ABB RobotStudio station: p3_Ejercicio_2018.rspag

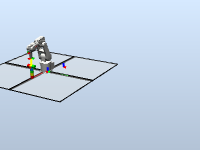
--- station ---
Station p3_Ejercicio_2018 (saved by RobotStudio 6.6.7701.1025)
Controller Sistema8
  mechanical unit ROB_1: IRB120_3_58__01_2, 6 joints, base frame (0, 0, 0) mm
Layout (positions relative to the parent item):
  - Grupo_1 [graphiccomponentgroup]
    - Pieza4 [part] at (170.19, 192.84, 150.02) mm, rotated rx 0 ry 0 rz -40 deg
    - Pieza3_2 [part] at (99.94, 75, 235.51) mm, rotated rx 90 ry 2 rz 0 deg
    - Pieza3 [part] at (100, 0, 100) mm
    - Pieza2_2 [part] at (99.94, 25, 235.51) mm, rotated rx 90 ry 2 rz 0 deg
    - Pieza2 [part] at (100, 0, 50.05) mm
    - Pieza1_2 [part] at (99.94, -25, 235.51) mm, rotated rx 90 ry 2 rz 0 deg
    - Pieza1 [part] at (100, 0, 0.18) mm
  - IRB120_3_58__01_2 [mechanism, from Robots\IRB120_3_58_G_01.rslib] at (0, 0, 0) mm; joint values [0, 0.3398, -0.1178, 0, 1.3488, 3.1416] (rad or m)
  - SC_Ventosa2 [smart component]
      signals: DI vacio, DI soplado, DO Vacuostato
      connections:
        SC_Ventosa.Vacuostato -> SC_Ventosa2.Vacuostato
        SC_Ventosa2.vacio -> SC_Ventosa.vacio
        SC_Ventosa2.soplado -> SC_Ventosa.soplado
    - SC_Ventosa [smart component] at (0, 0, 0) mm
        signals: DI vacio, DI soplado, DO Vacuostato
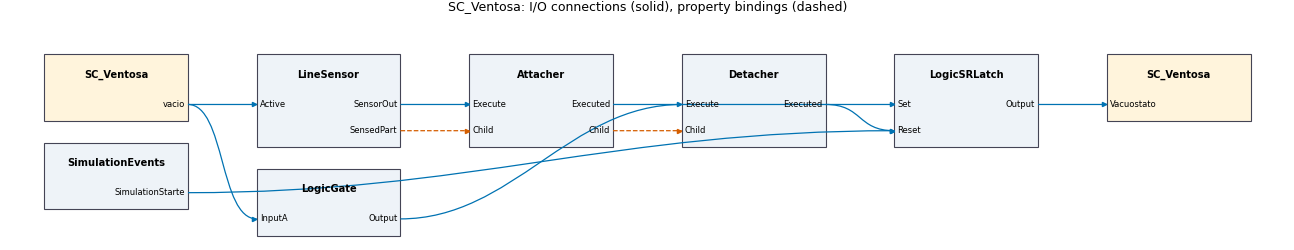
        connections:
          SC_Ventosa.vacio -> LineSensor.Active
          LineSensor.SensorOut -> Attacher.Execute
          Attacher.Executed -> LogicSRLatch.Set
          LogicSRLatch.Output -> SC_Ventosa.Vacuostato
          SC_Ventosa.vacio -> LogicGate.InputA
          LogicGate.Output -> Detacher.Execute
          Detacher.Executed -> LogicSRLatch.Reset
          SimulationEvents.SimulationStarted -> LogicSRLatch.Reset
          LineSensor.SensedPart => Attacher.Child
          Attacher.Child => Detacher.Child
      - MyNewTool [mechanism] at (400, 0, 474.33) mm, rotated rx -180 ry 0 rz 0 deg
          TCP Ventosa at (0, 0, 100) mm, rotated rx 180 ry 0 rz 0 deg
          links: Ventosa
      - LineSensor [smart component, from Components\LineSensor.rslib] at (400, 0, 474.33) mm, rotated rx -180 ry 0 rz 0 deg
          properties: Start=[0 0 0.0991]; End=[0 0 0.12]; Radius=0.002; SensedPart=Pieza1_2; SensedPoint=[0.4 -0.0750000686645508 0.231999969482422]
        - _sensorPart_ [part]
      - Attacher [smart component, from Components\Attacher.rslib]
          properties: Parent=MyNewTool; Flange=0; Child=Pieza1_2; Mount=false; Offset=[0 0 0]; Orientation=[0 0 0]
      - Detacher [smart component, from Components\Detacher.rslib]
          properties: Child=Pieza1_2; KeepPosition=true
      - LogicSRLatch [smart component, from Components\LogicSRLatch.rslib]
      - LogicGate [smart component, from Components\LogicGate.rslib]
          properties: Operator=NOT; Delay=0
      - SimulationEvents [smart component, from Components\SimulationEvents.rslib]
Attachment: MyNewTool is attached to IRB120_3_58__01_2 / Link6
Attachment: LineSensor is attached to MyNewTool / Ventosa
Station logic (signal -> signal, property => property):
  SC_Ventosa2.Vacuostato -> Sistema8.Vacuostado
  Sistema8.vacio -> SC_Ventosa2.vacio
  Sistema8.soplado -> SC_Ventosa2.soplado

--- Backups/Sistema8/RAPID/TASK1/PROGMOD/CalibData.mod ---
MODULE CalibData
	PERS tooldata Ventosa:=[TRUE,[[0.000043514,0,100],[0,1,0,-0.000000126]],[1,[0.000025299,0,100],[1,0,0,0],0,0,0]];
ENDMODULE

--- Backups/Sistema8/RAPID/TASK1/PROGMOD/Module1.mod ---
MODULE Module1
	CONST robtarget Target_10:=[[400.000012438,0,374.334869531],[1,0,-0.000000093,-0.000000044],[0,0,2,0],[9E+09,9E+09,9E+09,9E+09,9E+09,9E+09]];
	CONST robtarget Target_20:=[[400,0,200],[1,0,0,0],[0,0,1,0],[9E+09,9E+09,9E+09,9E+09,9E+09,9E+09]];
	CONST robtarget Target_30:=[[90.077,394.84,0],[1,0,0,0],[0,0,2,0],[9E+09,9E+09,9E+09,9E+09,9E+09,9E+09]];
    CONST robtarget Target_40:=[[-6.960015192,400.000008696,149.999960784],[0.694658412,0.000000021,-0.000000021,0.71933976],[1,-1,1,0],[9E+09,9E+09,9E+09,9E+09,9E+09,9E+09]];

	PROC Path_10()
        VAR robtarget reposo;
        VAR robtarget reposo1;
        VAR robtarget reposo2;
        VAR robtarget reposo3;
        VAR robtarget reposo4;

        VAR robtarget aux1;
        VAR robtarget aux2;
        VAR robtarget aux3;
        VAR robtarget aux4;




        reposo := Offs(Target_30,0,0,300);
        reposo1 := Offs(Target_30,0,0,50);
        reposo2 := Offs(Target_30,0,0,100);
        reposo3 := Offs(Target_30,0,0,150);
        reposo4 := Offs(Target_30,0,0,200);

        aux1 := Offs(Target_20,0,0,-50);
        aux2 := Offs(Target_20,0,0,-100);
        aux3 := Offs(Target_20,0,0,-150);
        aux4 := Offs(Target_20,0,0,-200);




        !Voy a inicio
	    MoveL Target_10,v1000,z100,Ventosa\WObj:=wobj0;
	    WaitTime 1;
        !Cojo la 1 pieza
	    MoveL Target_20,v1000,fine,Ventosa\WObj:=wobj0;
        WaitTime 1;
        SetDO vacio,1;
        WaitTime 1;
        !La dejo en posicion de reposo
        MoveJ reposo,v1000,fine,Ventosa\WObj:=wobj0;
	    MoveL reposo1,v500,fine,Ventosa\WObj:=wobj0;
        WaitTime 1;
	    SetDO vacio,0;
        WaitTime 1;
        !Vuelvo a inicio
        MoveJ Target_10,v1000,fine,Ventosa\WObj:=wobj0;

        !Cojo la 2 pieza
	    MoveL aux1,v1000,fine,Ventosa\WObj:=wobj0;
        WaitTime 1;
        SetDO vacio,1;
        WaitTime 1;
        !La dejo en posicion de reposo
        MoveJ reposo,v1000,fine,Ventosa\WObj:=wobj0;
	    MoveL reposo2,v500,fine,Ventosa\WObj:=wobj0;
	    SetDO vacio,0;
        WaitTime 1;
        !Vuelvo a inicio
        MoveJ Target_10,v1000,fine,Ventosa\WObj:=wobj0;

        !Cojo la 3 pieza
	    WaitTime 1;
	    MoveJ Target_10,v1000,fine,Ventosa\WObj:=wobj0;
	    MoveL aux2,v1000,fine,Ventosa\WObj:=wobj0;
        WaitTime 1;
        SetDO vacio,1;
        WaitTime 1;
        !La dejo en posicion de reposo
        MoveJ reposo,v1000,fine,Ventosa\WObj:=wobj0;
	    MoveL reposo3,v500,fine,Ventosa\WObj:=wobj0;
	    SetDO vacio,0;
        WaitTime 1;
        !Vuelvo a inicio
        MoveJ Target_10,v1000,fine,Ventosa\WObj:=wobj0;

        !Cojo la 4 pieza
	    MoveL aux3,v1000,fine,Ventosa\WObj:=wobj0;
        WaitTime 1;
        SetDO vacio,1;
        WaitTime 1;
        !La dejo en posicion de reposo
        MoveJ reposo,v1000,fine,Ventosa\WObj:=wobj0;
	    MoveL reposo4,v500,fine,Ventosa\WObj:=wobj0;
	    SetDO vacio,0;
        WaitTime 1;
        !Vuelvo a inicio
        MoveJ Target_10,v1000,fine,Ventosa\WObj:=wobj0;



        !Ahora las vuelvo a colocar.

        !Cojo la 4 pieza
	    MoveL reposo4,v1000,fine,Ventosa\WObj:=wobj0;
        WaitTime 1;
        SetDO vacio,1;
        WaitTime 1;
        !La dejo en posicion de reposo
        MoveJ Target_10,v1000,fine,Ventosa\WObj:=wobj0;
	    MoveL aux3,v500,fine,Ventosa\WObj:=wobj0;
	    SetDO vacio,0;
        WaitTime 1;
        !Vuelvo a inicio
        MoveJ Target_10,v1000,fine,Ventosa\WObj:=wobj0;

        !Cojo la 3 pieza
	    MoveL reposo3,v1000,fine,Ventosa\WObj:=wobj0;
        WaitTime 1;
        SetDO vacio,1;
        WaitTime 1;
        !La dejo en posicion de reposo
        MoveJ Target_10,v1000,fine,Ventosa\WObj:=wobj0;
	    MoveL aux2,v500,fine,Ventosa\WObj:=wobj0;
	    SetDO vacio,0;
        WaitTime 1;
        !Vuelvo a inicio
        MoveJ Target_10,v1000,fine,Ventosa\WObj:=wobj0;

        !Cojo la 2 pieza
	    MoveL reposo2,v1000,fine,Ventosa\WObj:=wobj0;
        WaitTime 1;
        SetDO vacio,1;
        WaitTime 1;
        !La dejo en posicion de reposo
        MoveJ Target_10,v1000,fine,Ventosa\WObj:=wobj0;
	    MoveL aux1,v500,fine,Ventosa\WObj:=wobj0;
	    SetDO vacio,0;
        WaitTime 1;
        !Vuelvo a inicio
        MoveJ Target_10,v1000,fine,Ventosa\WObj:=wobj0;

        !Cojo la 1 pieza
	    MoveL reposo1,v1000,fine,Ventosa\WObj:=wobj0;
        WaitTime 1;
        SetDO vacio,1;
        WaitTime 1;
        !La dejo en posicion de reposo
        MoveJ Target_10,v1000,fine,Ventosa\WObj:=wobj0;
	    MoveL Target_20,v500,fine,Ventosa\WObj:=wobj0;
	    SetDO vacio,0;
        !Vuelvo a inicio
        MoveJ Target_10,v1000,fine,Ventosa\WObj:=wobj0;




	ENDPROC

PROC piezagir()
        VAR robtarget p2_1;
        VAR robtarget p2_2;
        VAR robtarget p2_3;
        VAR robtarget a1_gir;
        VAR robtarget a2_gir;
        VAR robtarget a3_gir;
        VAR robtarget a3_gir_aux;
        VAR robtarget colision;

        a1_gir := RelTool(Target_20,0,-25,32, \Rx:=90);
        a2_gir := Offs(a1_gir,0,-50,0);

        a3_gir := Offs(a1_gir,0,50,0);



        colision := Offs (Target_10,0,-100,-50);
        p2_1  := Target_40;
        p2_2 := Offs(Target_40,0,0,-50);
        p2_3 := Offs(Target_40,0,0,-100);





        !Cojo la 1 pieza
	    MoveL p2_1,v1000,fine,Ventosa\WObj:=wobj0;
        WaitTime 1;
        SetDO vacio,1;
        WaitTime 1;
        !La dejo en posicion de reposo
	    MoveL a3_gir,v200,fine,Ventosa\WObj:=wobj0;
        WaitTime 1;
	    SetDO vacio,0;
        WaitTime 1;
        !Vuelvo a inicio
        MoveJ Target_10,v1000,fine,Ventosa\WObj:=wobj0;


        !Cojo la 2 pieza
	    MoveL p2_2,v1000,fine,Ventosa\WObj:=wobj0;
        WaitTime 1;
        SetDO vacio,1;
        WaitTime 1;
        MoveJ Target_10,v1000,fine,Ventosa\WObj:=wobj0;
        MoveJ colision,v1000,fine,Ventosa\WObj:=wobj0;
        !La dejo en posicion de reposo
	    MoveJ a1_gir,v200,fine,Ventosa\WObj:=wobj0;
        WaitTime 1;
	    SetDO vacio,0;
        WaitTime 1;
        !Vuelvo a inicio
        MoveJ Target_10,v1000,fine,Ventosa\WObj:=wobj0;

                !Cojo la 3 pieza
	    MoveL p2_3,v1000,fine,Ventosa\WObj:=wobj0;
        WaitTime 1;
        SetDO vacio,1;
        WaitTime 1;
        MoveJ Target_10,v1000,fine,Ventosa\WObj:=wobj0;
        MoveJ colision,v1000,fine,Ventosa\WObj:=wobj0;
        !La dejo en posicion de reposo
	    MoveL a2_gir,v200,fine,Ventosa\WObj:=wobj0;
        WaitTime 1;
	    SetDO vacio,0;
        WaitTime 1;
        !Vuelvo a inicio
        MoveJ Target_10,v1000,fine,Ventosa\WObj:=wobj0;









ENDPROC



	PROC main()
        Path_10;
	    piezagir;
	ENDPROC


ENDMODULE

--- Backups/Sistema8/RAPID/TASK1/SYSMOD/LINKEDM.sys ---
%%%
  VERSION:1
  LANGUAGE:ENGLISH
%%%

MODULE LINKEDM (SYSMODULE)

! FOLLOWER
!     Name of electronically linked follower axis used by operator at teach pendent.
      PERS string l_f_axis_name{5}       :=  ["",  "", "", "", ""];

!     Name of the mechanical unit for follower axis.
      PERS string l_f_mecunt_n{5}  :=  ["", "", "", "", ""];

!     Linked follower axis number in the mechanical unit (first axis in mech. unit is number 1).
      PERS num l_f_axis_no{5}      :=  [0,          0,   0,  0,  0];

! MASTER
!     Name of the mechanical unit for linked master axis.
      PERS string l_m_mecunt_n{5} :=  ["", "", "", "", ""];

!     Linked master axis number in the mechanical unit (first axis in mech. unit is number 1).
!     See axis number table in documentation for different master mechanical units.
      PERS num l_m_axis_no{5}     :=  [0,  0,  0,  0,  0];

! POSITION OFFSET
!     The increase of the allowed offset position between the master and follower
!     positions, used when starting AUTO mode. As soon as the offset is decreased
!     the old configurated parameter is used.
!     Example: 3 => the configurated value of allowed offset is increased 3 times.
      PERS num offset_ratio{5}       :=  [10,  10,   10,  10,  10];

! SPEED RATIO
!     Speed_ratio used in AUTO and JOG modes [ very_slow   slow    normal    fast]
!     Value 1 = max allowed manual speed.
      CONST num speed_ratio {20}      := [0.01, 0.01, 0.01, 0.01, 0.01,
                                          0.05, 0.05, 0.05, 0.05, 0.05,
                                          0.20, 0.20, 0.20, 0.20, 0.20,
                                          1.00, 1.00, 1.00, 1.00, 1.00];

! STEP SIZE
!     Displacement position used in JOG mode for each activation of positive or
!     negative movement.                  [very_short    short   normal   long]
!     Unit degees or meter.
      CONST num displacement {20}     := [0.001, 0.001, 0.001, 0.001, 0.001,
                                          0.005, 0.005, 0.005, 0.005, 0.005,
                                          0.020, 0.020, 0.020, 0.020, 0.020,
                                          0.100, 0.100, 0.100, 0.100, 0.100];


!-------------------------------------------------------------
 PROC Linked_m ()
      Linked_m_exe ;
 ENDPROC
ENDMODULE

--- Backups/Sistema8/SYSPAR/EIO.cfg ---
EIO:CFG_1.0:6:1::
#
INDUSTRIAL_NETWORK:

      -Name "DeviceNet" -Label "DeviceNet Master/Slave Network" -Address "2"\
      -Simulated
#
DEVICENET_DEVICE:

      -Name "ModuloES" -Simulated
#
DEVICENET_INTERNAL_DEVICE:

      -Name "DN_Internal_Device" -VendorName "ABB Robotics"\
      -ProductName "DeviceNet Internal Slave Device"
#
EIO_SIGNAL:

      -Name "vacio" -SignalType "DO" -Device "ModuloES" -DeviceMap "0"\
      -Category "vacio" -Access "All"

      -Name "soplado" -SignalType "DO" -Device "ModuloES" -Label "soplado"\
      -DeviceMap "1" -Access "All"

      -Name "Vacuostado" -SignalType "DI" -Device "ModuloES" -Label "Vacuostado"\
      -DeviceMap "0" -Access "All"
